{attribute 'qualified_only'}
(**VAR_GLOBAL PERSISTENT
	udi_Station_In_Error			:UDINT;
	udi_Station_In_Error_Code		:UDINT;
	ws_Stasion_In_Error				:WSTRING;
	ws_Station_Error_Description		:WSTRING(255);
	ws_Station_Error_Description_2	:WSTRING(255);
	A_Error_station	:ARRAY[0..100] OF ST_Error_Station_Handling; 
	A_Error_description	:ARRAY[0..500] OF ST_Error_Description_Handling;
	
	b_empy_error					:BOOL;
	b_new_system					:BOOL;
	
	sVisGuid						:STRING;
	
	b_reset_event_logger :BOOL;
END_VAR**)
VAR_GLOBAL
	b_reset_event_logger :BOOL;
	logowanie_krok: INT;
	b_cameras_ivms:BOOL;
END_VAR

(* stored: Version 1.1.0.1, ProductVersion 3.1.4026.13, FileIdentifier 3bac60c7979e19e3b4c90357e10333a55778cd55, FileSignature 6119db199b4377b81c03a5a20033f20d94dbe35d9c377696eae1070653e130c0765e54bedb2bda108425c1e5283474d5249537c7b5398e2afb89e6ee891d1185b3116a7a2d39b0df3f57ccdbd6d7fdaaa444591aa1a88d67700484f6c64cdef0b890890c5359d2820298b6e39c155ffc43a16546008fce2f50fa5c81178cab1c35c024353fbaef407007cc0a30e4d20746e99787b90543ec97bb2793dcdec17f20a939d0e3b6fbe66c3c099652e9b394d1a643715ae4448d96e54e1ae443c69b598d547c4c31250d3d1aa5dbfbbf2faf1ae9f75cf6720fff77d5080e44d871db2ecc57283a017872440d4208bd357092f8812b01c27acbf462a7e3bfcb59dbc7
   GVL GVL_Error: Id {a6bf8a5a-690c-4b24-8a35-da0dcb8ed8de} *)
